(* PLC project Tennesee, Generated TextualNotationConverter 1.0 *)
(* stored: creationDateTime 2025-07-30T12:00:00, modificationDateTime 2025-09-18T08:11:10 *)

FUNCTION_BLOCK ANALOG_IN
  VAR_INPUT
    Name : STRING;
    Description : STRING;
    Raw_Signal : REAL;
    PV_High : REAL;
    PV_Low : REAL;
    Scaling_Slope : REAL;
    Scaling_Offset : REAL;
    Alarm_Enable : BOOL;
  END_VAR
  VAR_OUTPUT
    PV : REAL;
    High_Alarm : BOOL;
    Low_Alarm : BOOL;
    General_Fault : BOOL;
  END_VAR

            
          
END_FUNCTION_BLOCK

FUNCTION_BLOCK BOOL_IN
  VAR_INPUT
    Name : STRING;
    Description : STRING;
    Bool_In : BOOL;
    Alarm_OnTrue : BOOL;
    Alarm_OnFalse : BOOL;
    Latch_Enable : BOOL;
    Reset_Latch : BOOL;
  END_VAR
  VAR_OUTPUT
    Bool_Out : BOOL;
    Alarm_Active : BOOL;
    Latched_Status : BOOL;
  END_VAR

            
          
END_FUNCTION_BLOCK

FUNCTION_BLOCK DIGITAL_IN
  VAR_INPUT
    Name : STRING;
    Description : STRING;
    DI_Raw : BOOL;
    DebounceTime : STRING;
    EnableAlarm : BOOL;
  END_VAR
  VAR_OUTPUT
    DI_Out : BOOL;
    Fault_State : BOOL;
  END_VAR

            
          
END_FUNCTION_BLOCK

FUNCTION_BLOCK DUTY_STANDBY
  VAR_INPUT
    Name : STRING;
    Description : STRING;
    Enable : BOOL;
    StartRequest : BOOL;
    AlternateEnable : BOOL;
    ForcePumpA : BOOL;
    ForcePumpB : BOOL;
    DutyElapsed : BOOL;
    MinRunElapsed : BOOL;
    SwitchoverDelayElapsed : BOOL;
    StartTimeoutElapsed : BOOL;
    PumpA_RunFB : BOOL;
    PumpB_RunFB : BOOL;
    PumpA_Fault : BOOL;
    PumpB_Fault : BOOL;
    Reset : BOOL;
    Inhibit : BOOL;
  END_VAR
  VAR_OUTPUT
    CmdPumpA : BOOL;
    CmdPumpB : BOOL;
    ActiveIsA : BOOL;
    SwitchedDueToDuty : BOOL;
    SwitchedDueToFailure : BOOL;
    Alarm_FailedStart_A : BOOL;
    Alarm_FailedStart_B : BOOL;
    Alarm_NoAvailablePump : BOOL;
  END_VAR

            
          
END_FUNCTION_BLOCK

FUNCTION_BLOCK MOTOR_2SPD
  VAR_INPUT
    Name : STRING;
    Description : STRING;
    Start_Cmd : BOOL;
    Stop_Cmd : BOOL;
    Speed_High_Cmd : BOOL;
    Speed_Low_Cmd : BOOL;
    Inhibit : BOOL;
  END_VAR
  VAR_OUTPUT
    Motor_Start_Out : BOOL;
    FB_Running : BOOL;
    FB_Trip : BOOL;
    FB_HighSpeed : BOOL;
    FB_LowSpeed : BOOL;
    Alarm_Speed_Error : BOOL;
  END_VAR

            
          
END_FUNCTION_BLOCK

FUNCTION_BLOCK MOTOR_ON_OFF
  VAR_INPUT
    Name : STRING;
    Description : STRING;
    Start_Cmd : BOOL;
    Stop_Cmd : BOOL;
    Start_Delay : STRING;
    MinRunTime : STRING;
    Inhibit : BOOL;
  END_VAR
  VAR_OUTPUT
    Motor_Start_Out : BOOL;
    FB_Running : BOOL;
    FB_Trip : BOOL;
    Alarm_Start_Fail : BOOL;
    Alarm_Stop_Fail : BOOL;
  END_VAR

            
          
END_FUNCTION_BLOCK

FUNCTION_BLOCK MOTOR_VSD
  VAR_INPUT
    Name : STRING;
    Description : STRING;
    Start_Cmd : BOOL;
    Stop_Cmd : BOOL;
    Speed_SP : REAL;
    Accel_Ramp : STRING;
    Decel_Ramp : STRING;
    Inhibit : BOOL;
  END_VAR
  VAR_OUTPUT
    Speed_Out : REAL;
    FB_Running : BOOL;
    FB_Fault : BOOL;
    FB_Ready : BOOL;
    FB_ActualSpeed : REAL;
    Alarm_Speed_Deviation : BOOL;
    Alarm_Comm_Fail : BOOL;
  END_VAR

            
          
END_FUNCTION_BLOCK

FUNCTION_BLOCK PID_BASIC
  VAR_INPUT
    Name : STRING;
    Description : STRING;
    AUTO : BOOL;
    PV : REAL;
    SP : REAL;
    MV_MIN : REAL;
    MV_MAX : REAL;
    X0 : REAL;
    KP : REAL;
    TR : REAL;
    TD : REAL;
    PV_High : REAL;
    PV_Low : REAL;
    Deviation_Limit : REAL;
    Inhibit : BOOL;
  END_VAR
  VAR_OUTPUT
    PV_High_Alarm : BOOL;
    PV_Low_Alarm : BOOL;
    Deviation_Alarm : BOOL;
    XOUT : REAL;
  END_VAR

            
          
END_FUNCTION_BLOCK

FUNCTION_BLOCK RATIO_CONTROL
  VAR_INPUT
    Name : STRING;
    Description : STRING;
    Auto : BOOL;
    PrimaryPV : REAL;
    SecondaryPV : REAL;
    RatioSP : REAL;
    Bias : REAL;
    TrimKp : REAL;
    TrimTi : STRING;
    MV_MIN : REAL;
    MV_MAX : REAL;
    ManOut : REAL;
    Inhibit : BOOL;
  END_VAR
  VAR_OUTPUT
    SlaveSP : REAL;
    ActiveRatio : REAL;
    RatioErr : REAL;
  END_VAR

            
          
END_FUNCTION_BLOCK

FUNCTION_BLOCK SPLIT_RANGE
  VAR_INPUT
    Name : STRING;
    Description : STRING;
    IN : REAL;
    Split_Point : REAL;
    Output1_Start : REAL;
    Output1_End : REAL;
    Output2_Start : REAL;
    Output2_End : REAL;
  END_VAR
  VAR_OUTPUT
    OUT1 : REAL;
    OUT2 : REAL;
  END_VAR

            
          
END_FUNCTION_BLOCK

FUNCTION_BLOCK VALVE_ELECTRIC
  VAR_INPUT
    Name : STRING;
    Description : STRING;
    Control_Signal : REAL;
    Manual_Mode : BOOL;
    Manual_Position : REAL;
    Open_Limit : REAL;
    Close_Limit : REAL;
    Timeout : STRING;
    Inhibit : BOOL;
  END_VAR
  VAR_OUTPUT
    Valve_Position : REAL;
    Feedback_Pos : REAL;
    Valve_Moving : BOOL;
    Position_Error : BOOL;
    Alarm : BOOL;
  END_VAR

            
          
END_FUNCTION_BLOCK

FUNCTION_BLOCK VALVE_ON_OFF
  VAR_INPUT
    Name : STRING;
    Description : STRING;
    Open_Cmd : BOOL;
    Close_Cmd : BOOL;
    Timeout : STRING;
    Inhibit : BOOL;
  END_VAR
  VAR_OUTPUT
    FB_Opened : BOOL;
    FB_Closed : BOOL;
    Valve_Open_Out : BOOL;
    Valve_Close_Out : BOOL;
    Alarm_Position_Error : BOOL;
    Alarm_General : BOOL;
  END_VAR

            
          
END_FUNCTION_BLOCK

FUNCTION_BLOCK VOTING_ANALOG
  VAR_INPUT
    Name : STRING;
    Description : STRING;
    Input1 : REAL;
    Input2 : REAL;
    Input3 : REAL;
    Deviation_Limit : REAL;
    Voting_Scheme : STRING;
    EnableAlarm : BOOL;
    Inhibit : BOOL;
  END_VAR
  VAR_OUTPUT
    Voted_Output : REAL;
    Sensor1_Fault : BOOL;
    Sensor2_Fault : BOOL;
    Sensor3_Fault : BOOL;
    Alarm_Voting_Error : BOOL;
    Healthy_Sensors_Count : INT;
  END_VAR

            
          
END_FUNCTION_BLOCK

PROGRAM Sec2
  VAR
    FIT101_Flow_PV_GPM : REAL;
    PI001_Pressure_PV_psig : REAL;
    FIC104_MV_to_PV103_Pct : REAL;
  END_VAR
  VAR
    FIT-101 : ANALOG_IN;
    PI-001 : ANALOG_IN;
    FIC-104 : PID_BASIC;
    PV-103 : VALVE_ELECTRIC;
    XV-106 : VALVE_ON_OFF;
    IAL-101 : BOOL_IN;
    FAL-101 : DIGITAL_IN;
    FAL-102 : DIGITAL_IN;
    FAL-103 : DIGITAL_IN;
  END_VAR

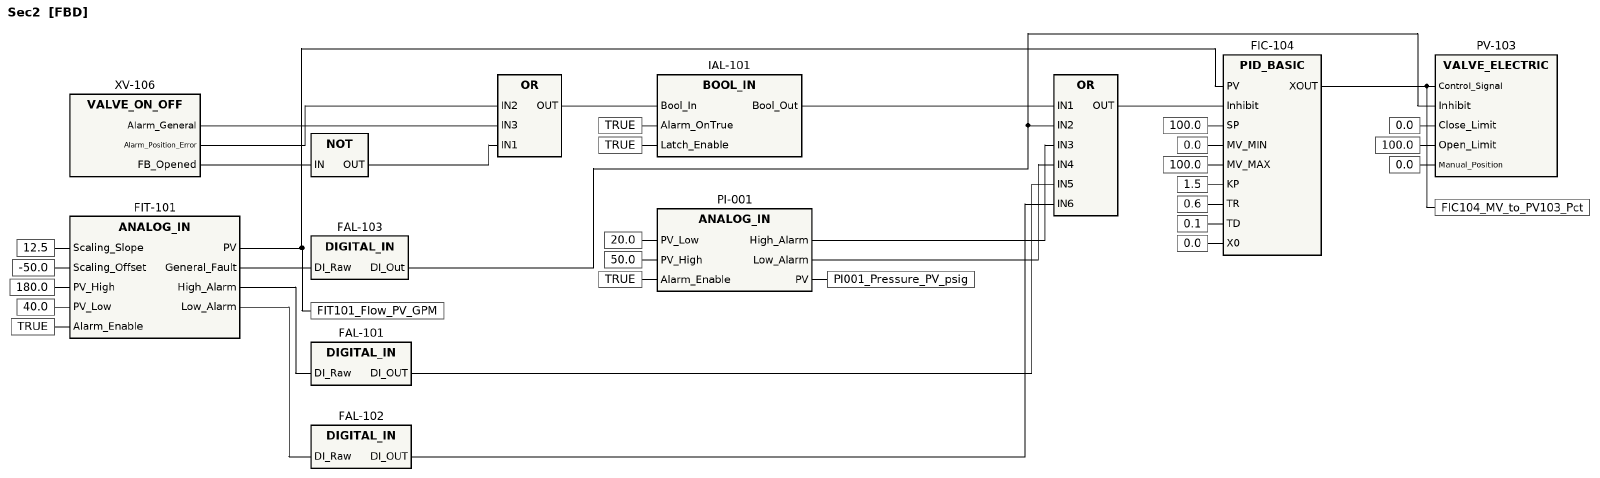
(* FBD diagram, written out as Structured Text *)
FIT-101(Scaling_Slope := 12.5, Scaling_Offset := -50.0, PV_High := 180.0, PV_Low := 40.0, Alarm_Enable := TRUE);
XV-106();
IAL-101(Bool_In := XV-106.Alarm_Position_Error OR XV-106.Alarm_General OR NOT XV-106.FB_Opened, Alarm_OnTrue := TRUE, Latch_Enable := TRUE);
FAL-103(DI_Raw := FIT-101.General_Fault);
PI-001(PV_Low := 20.0, PV_High := 50.0, Alarm_Enable := TRUE);
FAL-101(DI_Raw := FIT-101.High_Alarm);
FAL-102(DI_Raw := FIT-101.Low_Alarm);
FIC-104(PV := FIT-101.PV, Inhibit := IAL-101.Bool_Out OR FAL-103.DI_Out OR PI-001.High_Alarm OR PI-001.Low_Alarm OR FAL-101.DI_OUT OR FAL-102.DI_OUT, SP := 100.0, MV_MIN := 0.0, MV_MAX := 100.0, KP := 1.5, TR := 0.6, TD := 0.1, X0 := 0.0);
FIC104_MV_to_PV103_Pct := FIC-104.XOUT;
FIT101_Flow_PV_GPM := FIT-101.PV;
PI001_Pressure_PV_psig := PI-001.PV;
PV-103(Control_Signal := FIC-104.XOUT, Inhibit := FAL-103.DI_Out, Close_Limit := 0.0, Open_Limit := 100.0, Manual_Position := 0.0);
END_PROGRAM

PROGRAM Sec3
  VAR
    TIT-103_Temperature_C : REAL;
    LT-105_Level_Percent : REAL;
    TIC-101_Output_Percent : REAL;
    LIC-106_Output_Percent : REAL;
  END_VAR
  VAR
    TIT-103 : ANALOG_IN;
    LT-105 : ANALOG_IN;
    TIC-101 : PID_BASIC;
    LIC-106 : PID_BASIC;
    FC-004 : PID_BASIC;
    LV-104 : VALVE_ELECTRIC;
    XV-102 : VALVE_ON_OFF;
  END_VAR

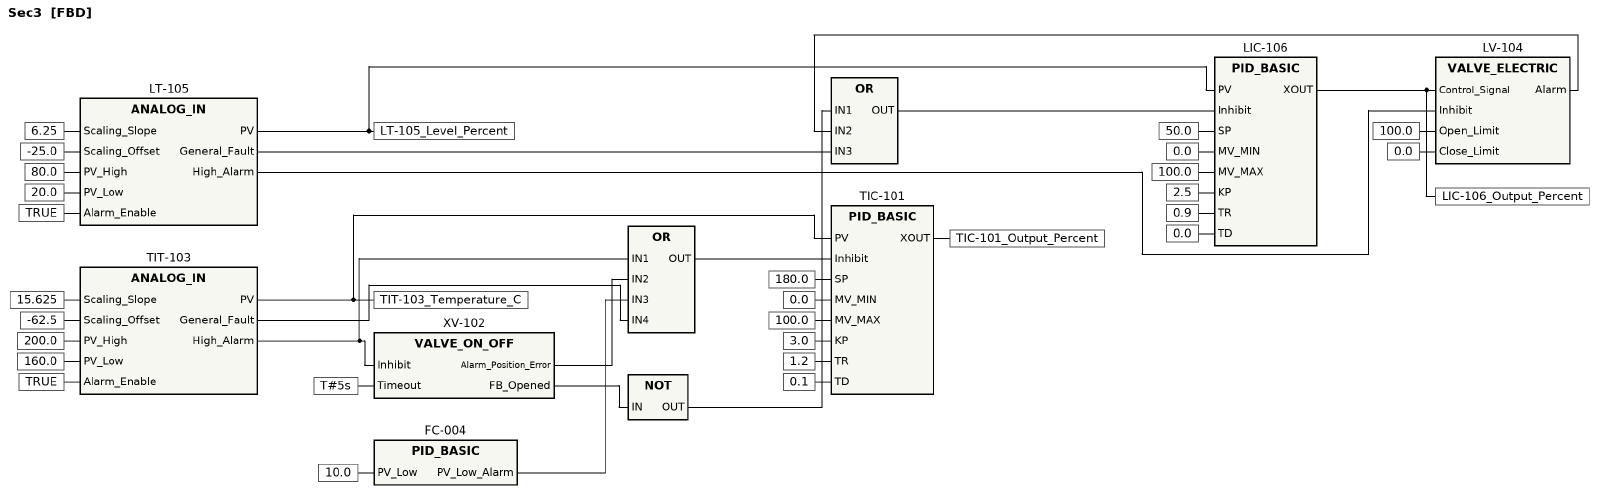
(* FBD diagram, written out as Structured Text *)
LT-105(Scaling_Slope := 6.25, Scaling_Offset := -25.0, PV_High := 80.0, PV_Low := 20.0, Alarm_Enable := TRUE);
TIT-103(Scaling_Slope := 15.625, Scaling_Offset := -62.5, PV_High := 200.0, PV_Low := 160.0, Alarm_Enable := TRUE);
XV-102(Inhibit := TIT-103.High_Alarm, Timeout := T#5s);
LV-104(Control_Signal := LIC-106.XOUT, Inhibit := LT-105.High_Alarm, Open_Limit := 100.0, Close_Limit := 0.0);
LIC-106(PV := LT-105.PV, Inhibit := NOT XV-102.FB_Opened OR LV-104.Alarm OR LT-105.General_Fault, SP := 50.0, MV_MIN := 0.0, MV_MAX := 100.0, KP := 2.5, TR := 0.9, TD := 0.0);
LIC-106_Output_Percent := LIC-106.XOUT;
LT-105_Level_Percent := LT-105.PV;
FC-004(PV_Low := 10.0);
TIC-101(PV := TIT-103.PV, Inhibit := TIT-103.High_Alarm OR XV-102.Alarm_Position_Error OR FC-004.PV_Low_Alarm OR TIT-103.General_Fault, SP := 180.0, MV_MIN := 0.0, MV_MAX := 100.0, KP := 3.0, TR := 1.2, TD := 0.1);
TIC-101_Output_Percent := TIC-101.XOUT;
TIT-103_Temperature_C := TIT-103.PV;
END_PROGRAM

PROGRAM Sec4
  VAR
    FIT103_FlowRate : REAL;
    LT104_Level : REAL;
    LIC101_PV102_ValveCommand : REAL;
    LAH101_Alarm : BOOL;
    LAL101_Alarm : BOOL;
    LT104_FaultAlarm : BOOL;
    OverCapacity_Active : BOOL;
    LevelAbove10_OK : BOOL;
  END_VAR
  VAR
    FIT-103 : ANALOG_IN;
    LT-104 : ANALOG_IN;
    LIC-101 : PID_BASIC;
    PV-102 : VALVE_ELECTRIC;
  END_VAR
  VAR  (* added by the conversion: wires and edge detectors of the diagram *)
    _GT146_OUT : BOOL;
    _GT148_OUT : BOOL;
  END_VAR

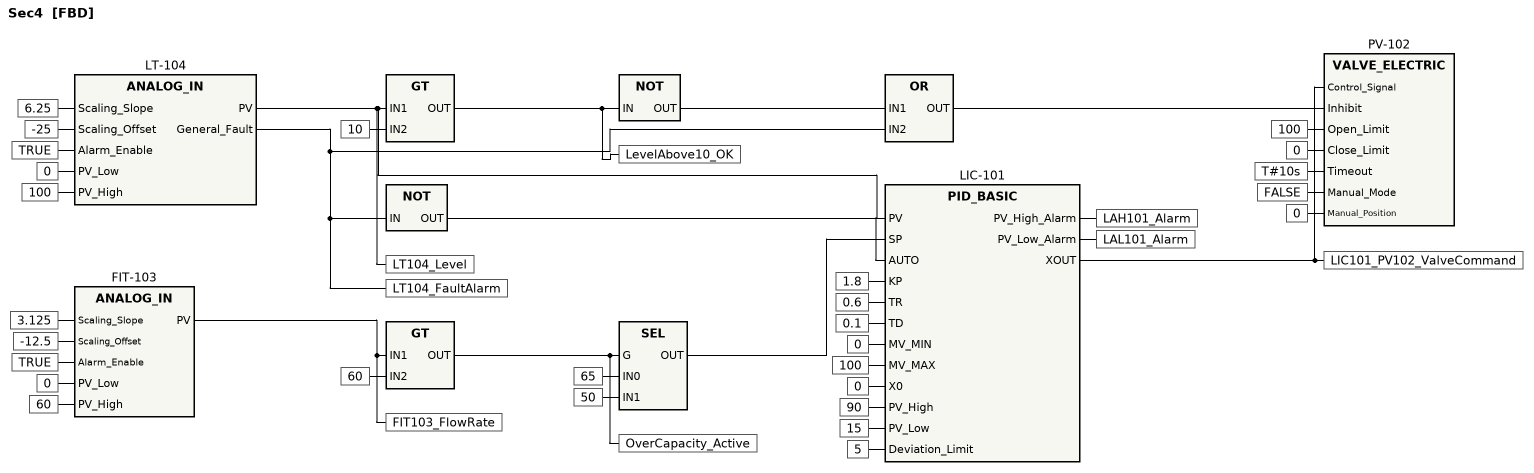
(* FBD diagram, written out as Structured Text *)
FIT-103(Scaling_Slope := 3.125, Scaling_Offset := -12.5, Alarm_Enable := TRUE, PV_Low := 0, PV_High := 60);
FIT103_FlowRate := FIT-103.PV;
LT-104(Scaling_Slope := 6.25, Scaling_Offset := -25, Alarm_Enable := TRUE, PV_Low := 0, PV_High := 100);
_GT146_OUT := FIT-103.PV > 60;
LIC-101(PV := LT-104.PV, SP := SEL(_GT146_OUT, 65, 50), AUTO := NOT LT-104.General_Fault, KP := 1.8, TR := 0.6, TD := 0.1, MV_MIN := 0, MV_MAX := 100, X0 := 0, PV_High := 90, PV_Low := 15, Deviation_Limit := 5);
LAH101_Alarm := LIC-101.PV_High_Alarm;
LAL101_Alarm := LIC-101.PV_Low_Alarm;
LIC101_PV102_ValveCommand := LIC-101.XOUT;
LT104_FaultAlarm := LT-104.General_Fault;
LT104_Level := LT-104.PV;
_GT148_OUT := LT-104.PV > 10;
LevelAbove10_OK := _GT148_OUT;
OverCapacity_Active := _GT146_OUT;
PV-102(Control_Signal := LIC-101.XOUT, Inhibit := NOT _GT148_OUT OR LT-104.General_Fault, Open_Limit := 100, Close_Limit := 0, Timeout := T#10s, Manual_Mode := FALSE, Manual_Position := 0);
END_PROGRAM

PROGRAM Sec5
  VAR
    TIT106_ReboilerTemp_PV : REAL;
    LT107_Column2Level_PV : REAL;
    TIC106_FV105_SteamFlow_MV : REAL;
    LIC107_LV102_Outflow_MV : REAL;
  END_VAR
  VAR
    TIT-106 : ANALOG_IN;
    LT-107 : ANALOG_IN;
    TIC-106 : PID_BASIC;
    LIC-107 : PID_BASIC;
    FV-105 : VALVE_ELECTRIC;
    LV-102 : VALVE_ELECTRIC;
    CONDENSATE_RETURN_VALVE_OPEN_LS : DIGITAL_IN;
  END_VAR

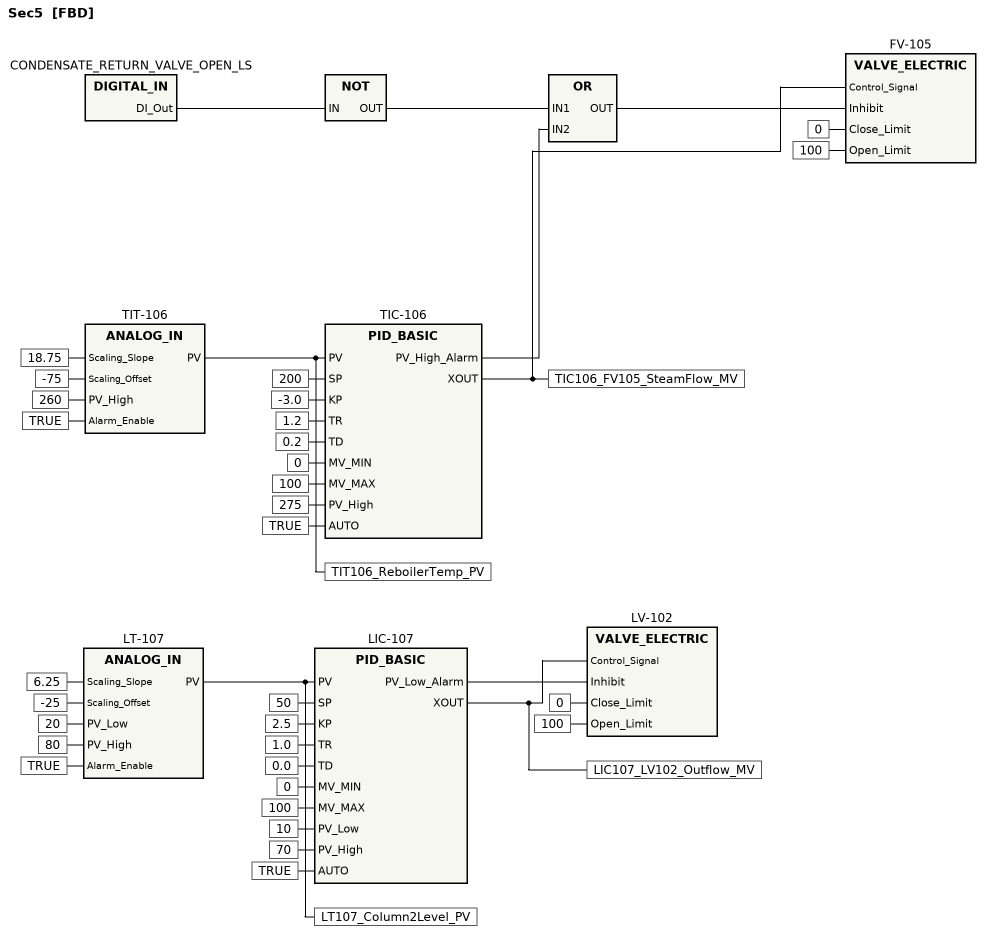
(* FBD diagram, written out as Structured Text *)
LT-107(Scaling_Slope := 6.25, Scaling_Offset := -25, PV_Low := 20, PV_High := 80, Alarm_Enable := TRUE);
LIC-107(PV := LT-107.PV, SP := 50, KP := 2.5, TR := 1.0, TD := 0.0, MV_MIN := 0, MV_MAX := 100, PV_Low := 10, PV_High := 70, AUTO := TRUE);
LIC107_LV102_Outflow_MV := LIC-107.XOUT;
LT107_Column2Level_PV := LT-107.PV;
TIT-106(Scaling_Slope := 18.75, Scaling_Offset := -75, PV_High := 260, Alarm_Enable := TRUE);
TIC-106(PV := TIT-106.PV, SP := 200, KP := -3.0, TR := 1.2, TD := 0.2, MV_MIN := 0, MV_MAX := 100, PV_High := 275, AUTO := TRUE);
TIC106_FV105_SteamFlow_MV := TIC-106.XOUT;
TIT106_ReboilerTemp_PV := TIT-106.PV;
CONDENSATE_RETURN_VALVE_OPEN_LS();
FV-105(Control_Signal := TIC-106.XOUT, Inhibit := NOT CONDENSATE_RETURN_VALVE_OPEN_LS.DI_Out OR TIC-106.PV_High_Alarm, Close_Limit := 0, Open_Limit := 100);
LV-102(Control_Signal := LIC-107.XOUT, Inhibit := LIC-107.PV_Low_Alarm, Close_Limit := 0, Open_Limit := 100);
END_PROGRAM

PROGRAM Sec7
  VAR
    TI_008_Temp_PV : REAL;
    LI_003_Level_PV : REAL;
    TIC_106_MV_Pct : REAL;
    LIC_103_MV_Pct : REAL;
    XV_105_Valve_Position_Pct : REAL;
    XV_104_Valve_Position_Pct : REAL;
    Column3_Start_CMD : BOOL;
    TIC106_DeviationFault : BOOL;
    LIC101_Condensate_High : BOOL;
  END_VAR
  VAR
    LI-003 : ANALOG_IN;
    TI-008 : ANALOG_IN;
    LIC-103 : PID_BASIC;
    TIC-106 : PID_BASIC;
    XV-104 : VALVE_ELECTRIC;
    XV-105 : VALVE_ELECTRIC;
    LIC-101-HI : BOOL_IN;
  END_VAR
  VAR  (* added by the conversion: wires and edge detectors of the diagram *)
    _OR244_OUT : BOOL;
    _OR236_OUT : BOOL;
  END_VAR

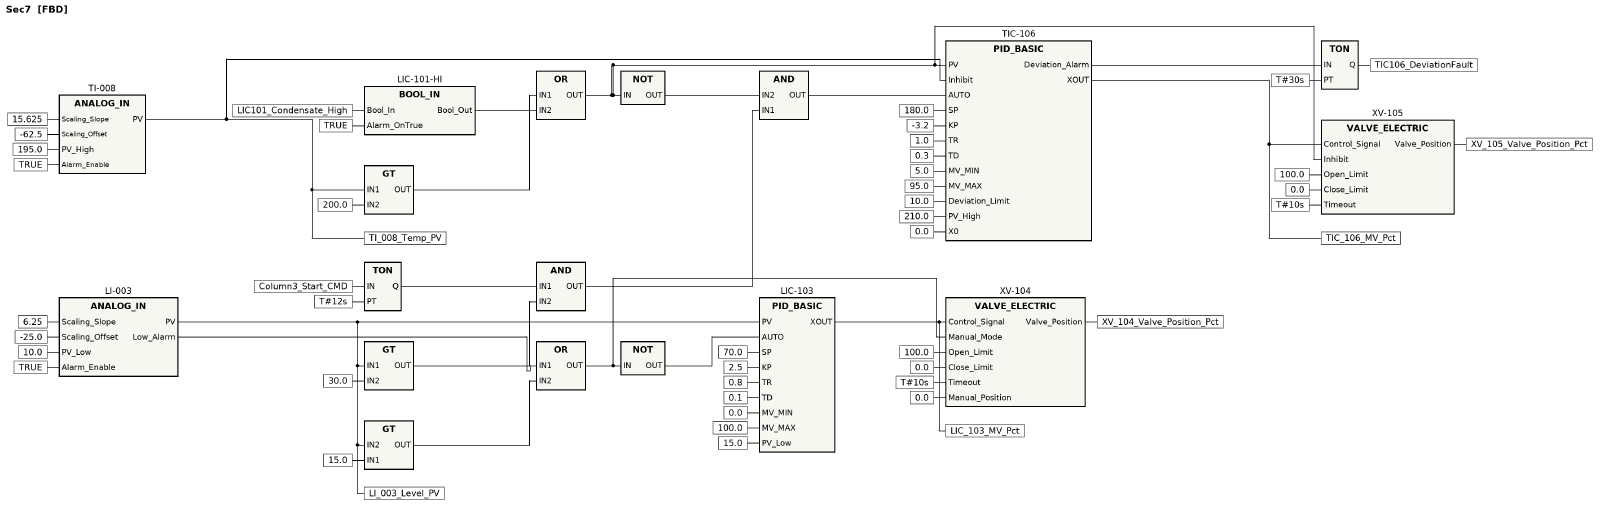
(* FBD diagram, written out as Structured Text *)
LI-003(Scaling_Slope := 6.25, Scaling_Offset := -25.0, PV_Low := 10.0, Alarm_Enable := TRUE);
_OR244_OUT := LI-003.Low_Alarm OR LI-003.PV > 15.0;
LIC-103(PV := LI-003.PV, AUTO := NOT _OR244_OUT, SP := 70.0, KP := 2.5, TR := 0.8, TD := 0.1, MV_MIN := 0.0, MV_MAX := 100.0, PV_Low := 15.0);
LIC_103_MV_Pct := LIC-103.XOUT;
LI_003_Level_PV := LI-003.PV;
TI-008(Scaling_Slope := 15.625, Scaling_Offset := -62.5, PV_High := 195.0, Alarm_Enable := TRUE);
LIC-101-HI(Bool_In := LIC101_Condensate_High, Alarm_OnTrue := TRUE);
_OR236_OUT := TI-008.PV > 200.0 OR LIC-101-HI.Bool_Out;
TIC-106(PV := TI-008.PV, Inhibit := _OR236_OUT, AUTO := NOT _OR236_OUT AND TON(Column3_Start_CMD, T#12s) AND LI-003.PV > 30.0, SP := 180.0, KP := -3.2, TR := 1.0, TD := 0.3, MV_MIN := 5.0, MV_MAX := 95.0, Deviation_Limit := 10.0, PV_High := 210.0, X0 := 0.0);
TIC106_DeviationFault := TON(TIC-106.Deviation_Alarm, T#30s);
TIC_106_MV_Pct := TIC-106.XOUT;
TI_008_Temp_PV := TI-008.PV;
XV-104(Control_Signal := LIC-103.XOUT, Manual_Mode := _OR244_OUT, Open_Limit := 100.0, Close_Limit := 0.0, Timeout := T#10s, Manual_Position := 0.0);
XV_104_Valve_Position_Pct := XV-104.Valve_Position;
XV-105(Control_Signal := TIC-106.XOUT, Inhibit := _OR236_OUT, Open_Limit := 100.0, Close_Limit := 0.0, Timeout := T#10s);
XV_105_Valve_Position_Pct := XV-105.Valve_Position;
END_PROGRAM

PROGRAM Sec8
  VAR
    LT102_Level_PV_Pct : REAL;
    FIT105_Flow_PV_LPM : REAL;
    LIC106_MV_To_XV101_Pct : REAL;
    FC008_MV_To_PV104_Pct : REAL;
    Decanter2_Online : BOOL;
  END_VAR
  VAR
    FIT-105 : ANALOG_IN;
    LT-102 : ANALOG_IN;
    LT-103 : ANALOG_IN;
    LT-107 : ANALOG_IN;
    LIC-106 : PID_BASIC;
    FC-008 : PID_BASIC;
    XV-101 : VALVE_ELECTRIC;
    PV-104 : VALVE_ELECTRIC;
  END_VAR
  VAR  (* added by the conversion: wires and edge detectors of the diagram *)
    _LT311_OUT : BOOL;
    _OR317_OUT : BOOL;
    _OR303_OUT : BOOL;
  END_VAR

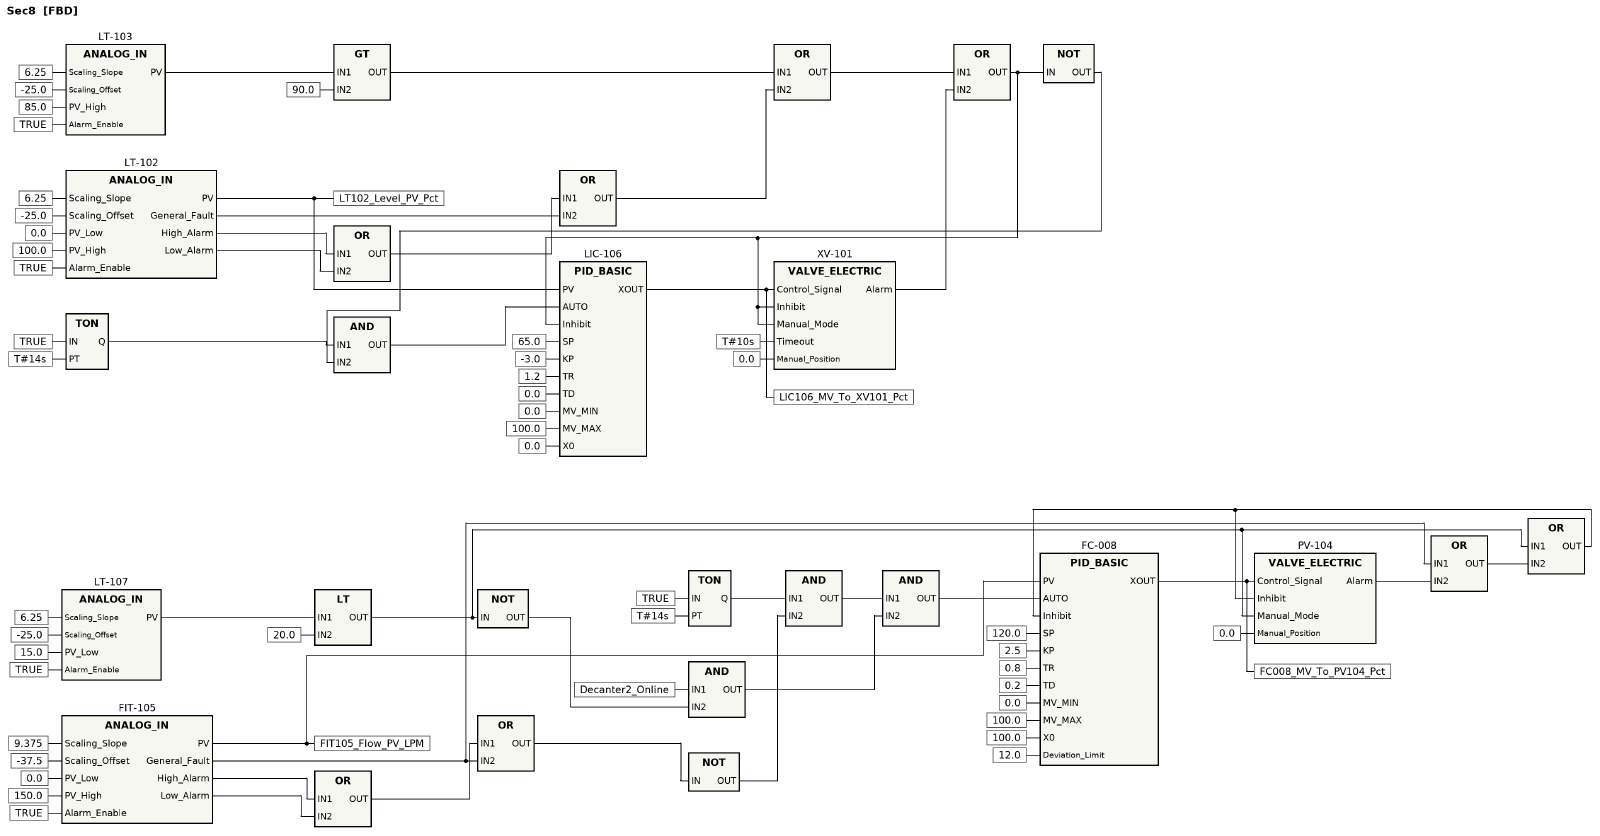
(* FBD diagram, written out as Structured Text *)
FIT-105(Scaling_Slope := 9.375, Scaling_Offset := -37.5, PV_Low := 0.0, PV_High := 150.0, Alarm_Enable := TRUE);
LT-107(Scaling_Slope := 6.25, Scaling_Offset := -25.0, PV_Low := 15.0, Alarm_Enable := TRUE);
_LT311_OUT := LT-107.PV < 20.0;
PV-104(Control_Signal := FC-008.XOUT, Inhibit := _OR317_OUT, Manual_Mode := _LT311_OUT, Manual_Position := 0.0);
_OR317_OUT := _LT311_OUT OR FIT-105.General_Fault OR PV-104.Alarm;
FC-008(PV := FIT-105.PV, AUTO := TON(TRUE, T#14s) AND NOT (FIT-105.High_Alarm OR FIT-105.Low_Alarm OR FIT-105.General_Fault) AND Decanter2_Online AND NOT _LT311_OUT, Inhibit := _OR317_OUT, SP := 120.0, KP := 2.5, TR := 0.8, TD := 0.2, MV_MIN := 0.0, MV_MAX := 100.0, X0 := 100.0, Deviation_Limit := 12.0);
FC008_MV_To_PV104_Pct := FC-008.XOUT;
FIT105_Flow_PV_LPM := FIT-105.PV;
LT-102(Scaling_Slope := 6.25, Scaling_Offset := -25.0, PV_Low := 0.0, PV_High := 100.0, Alarm_Enable := TRUE);
LT-103(Scaling_Slope := 6.25, Scaling_Offset := -25.0, PV_High := 85.0, Alarm_Enable := TRUE);
XV-101(Control_Signal := LIC-106.XOUT, Inhibit := _OR303_OUT, Manual_Mode := _OR303_OUT, Timeout := T#10s, Manual_Position := 0.0);
_OR303_OUT := LT-103.PV > 90.0 OR LT-102.High_Alarm OR LT-102.Low_Alarm OR LT-102.General_Fault OR XV-101.Alarm;
LIC-106(PV := LT-102.PV, AUTO := TON(TRUE, T#14s) AND NOT _OR303_OUT, Inhibit := _OR303_OUT, SP := 65.0, KP := -3.0, TR := 1.2, TD := 0.0, MV_MIN := 0.0, MV_MAX := 100.0, X0 := 0.0);
LIC106_MV_To_XV101_Pct := LIC-106.XOUT;
LT102_Level_PV_Pct := LT-102.PV;
END_PROGRAM

PROGRAM Sec9
  VAR
    TIT101_Temperature_PV_C : REAL;
    FI103_Flow_PV : REAL;
    FIC103_Output_MV_Percent : REAL;
    LV102_ValvePositionCmd_Percent : REAL;
    XV104_Open_FB : BOOL;
    LC002_ValidLevel : BOOL;
    LC002_LevelValid_In : BOOL;
  END_VAR
  VAR
    TIT-101 : ANALOG_IN;
    FI-103 : ANALOG_IN;
    FIC-103 : PID_BASIC;
    LV-102 : VALVE_ELECTRIC;
    XV-104 : VALVE_ON_OFF;
    LC-002 : BOOL_IN;
  END_VAR
  VAR  (* added by the conversion: wires and edge detectors of the diagram *)
    _NOT374_OUT : BOOL;
    _OR376_OUT : BOOL;
  END_VAR

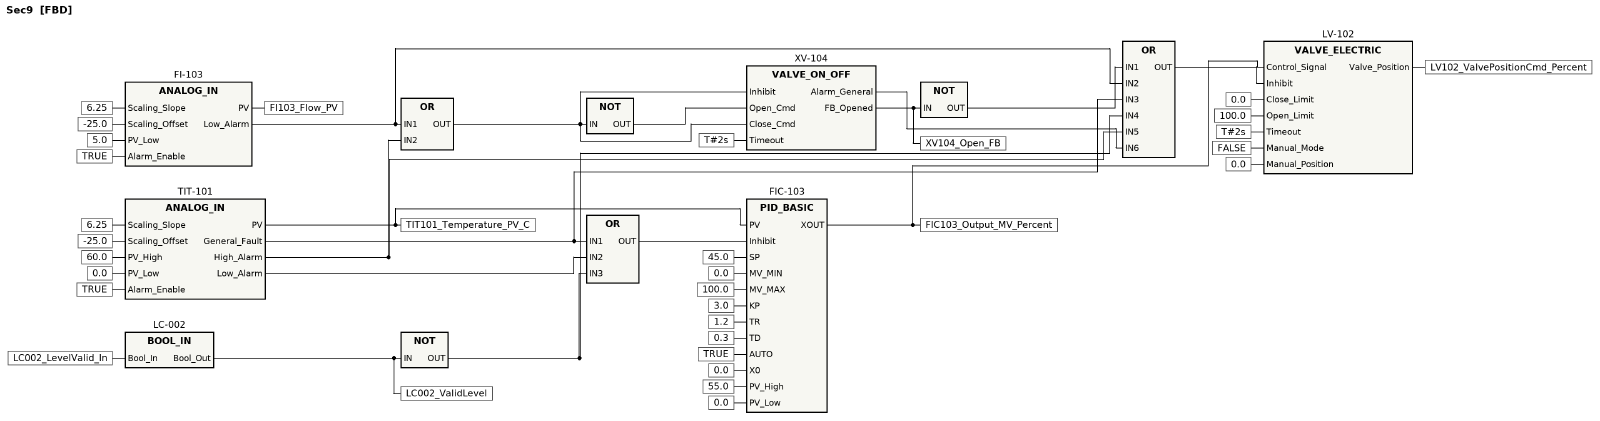
(* FBD diagram, written out as Structured Text *)
FI-103(Scaling_Slope := 6.25, Scaling_Offset := -25.0, PV_Low := 5.0, Alarm_Enable := TRUE);
FI103_Flow_PV := FI-103.PV;
TIT-101(Scaling_Slope := 6.25, Scaling_Offset := -25.0, PV_High := 60.0, PV_Low := 0.0, Alarm_Enable := TRUE);
LC-002(Bool_In := LC002_LevelValid_In);
_NOT374_OUT := NOT LC-002.Bool_Out;
FIC-103(PV := TIT-101.PV, Inhibit := TIT-101.General_Fault OR TIT-101.Low_Alarm OR _NOT374_OUT, SP := 45.0, MV_MIN := 0.0, MV_MAX := 100.0, KP := 3.0, TR := 1.2, TD := 0.3, AUTO := TRUE, X0 := 0.0, PV_High := 55.0, PV_Low := 0.0);
FIC103_Output_MV_Percent := FIC-103.XOUT;
LC002_ValidLevel := LC-002.Bool_Out;
_OR376_OUT := FI-103.Low_Alarm OR TIT-101.High_Alarm;
XV-104(Inhibit := _OR376_OUT, Open_Cmd := NOT _OR376_OUT, Close_Cmd := _OR376_OUT, Timeout := T#2s);
LV-102(Control_Signal := FIC-103.XOUT, Inhibit := NOT XV-104.FB_Opened OR FI-103.Low_Alarm OR TIT-101.General_Fault OR _NOT374_OUT OR TIT-101.High_Alarm OR XV-104.Alarm_General, Close_Limit := 0.0, Open_Limit := 100.0, Timeout := T#2s, Manual_Mode := FALSE, Manual_Position := 0.0);
LV102_ValvePositionCmd_Percent := LV-102.Valve_Position;
TIT101_Temperature_PV_C := TIT-101.PV;
XV104_Open_FB := XV-104.FB_Opened;
END_PROGRAM

CONFIGURATION Config0
  RESOURCE Res0 ON PLC
    TASK task0(INTERVAL := T#20ms, PRIORITY := 0);
    PROGRAM instance0 WITH task0 : Reviewed_out;
    PROGRAM instance_1 WITH task0 : Industrial Automation;
    PROGRAM instance_2 WITH task0 : Sec2;
    PROGRAM instance_3 WITH task0 : Sec3;
    PROGRAM instance_4 WITH task0 : Sec4;
    PROGRAM instance_5 WITH task0 : Sec5;
    PROGRAM instance_6 WITH task0 : Sec7;
    PROGRAM instance_7 WITH task0 : Sec8;
    PROGRAM instance_8 WITH task0 : Sec9;
  END_RESOURCE
END_CONFIGURATION
